(* IEC 61131-3 sources: plcassist-cli/packages/volt-lsp-iec/test-corpus/twincat-project14/GVLs, 1 file *)

(* ---- GVL_PackML.gvl ---- *)
{attribute 'qualified_only'}
VAR_GLOBAL CONSTANT
    UNIT_STATE_TIMEOUT_DEFAULT : TIME := T#10S;
END_VAR
VAR_GLOBAL
END_VAR
